DATA_BLOCK "ST10_Flow8_FRobot_2_iDB"
{ S7_Optimized_Access := 'TRUE' }
VERSION : 0.1
NON_RETAIN
"ST10_Flow8_FRobot_2"

BEGIN

END_DATA_BLOCK

